PROGRAM Example06_PhaseSynchronization
VAR
  otgTimeSync : Struckig.Otg(cycletime:=0.001, dofs:=3) := (
                  Synchronization := SynchronizationType.TimeSync,
                  CurrentPosition :=     [ 0.0, 0.0, 0.0 ],
                  TargetPosition :=      [ 1.0, -1.0, 2.0 ],
                  MaxVelocity :=         [ 1.0, 1.0, 1.0 ],
                  MaxAcceleration :=     [ 1.0, 1.0, 1.0 ],
                  MaxJerk :=             [ 1.0, 1.0, 1.0 ]
  ); 
  
  otgPhaseSync : Struckig.Otg(cycletime:=0.001, dofs:=3) := (
                  Synchronization := SynchronizationType.Phase,
                  CurrentPosition :=     [ 0.0, 0.0, 0.0 ],
                  TargetPosition :=      [ 1.0, -1.0, 2.0 ],
                  MaxVelocity :=         [ 1.0, 1.0, 1.0 ],
                  MaxAcceleration :=     [ 1.0, 1.0, 1.0 ],
                  MaxJerk :=             [ 1.0, 1.0, 1.0 ]
  ); 
END_VAR

otgTimeSync(EnableAutoPropagate := TRUE);
otgPhaseSync(EnableAutoPropagate := TRUE);

END_PROGRAM

(* stored: Version 1.1.0.1, ProductVersion 3.1.4024.9
   POU Example06_PhaseSynchronization: Id {4ad92911-ea39-417e-bb7d-fd1ee164d4a9}, SpecialFunc None *)
